ABB RobotStudio station: Assignment1 - Sela Shapira.rspag

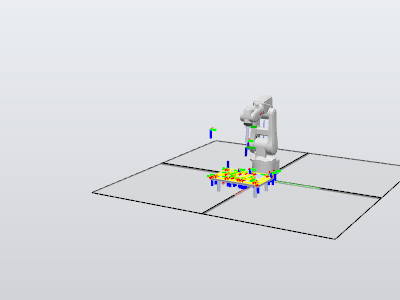
--- station ---
Station Assignment1 - Sela Shapira (saved by RobotStudio 23.2.10478.1)
Controller IRB120_3_58
  mechanical unit ROB_1: IRB120_3_58__01, 6 joints, base frame (0, 0, 0) mm
Layout (positions relative to the parent item):
  - IRB120_3_58__01 [mechanism, from %ABB.RobotStudio.Models.IRB120%\IRB120_3_58_G_01.rslib] at (0, 0, 0) mm; joint values [0.0316, -0.0225, 0.1697, 0.0059, 1.2834, -0.0224] (rad or m)
  - MyPen [mechanism, from Robotstudio\MyPen.rslib] at (312.81, 10.28, 513.58) mm, rotated rx 179.85 ry 8.04 rz -176.99 deg
  - A3 table [part] at (370, 0, 100) mm, rotated rx 90 ry 0 rz 90 deg, size 420 x 110 x 300 mm
  - Part_2 [part] at (370, 0, 100) mm, rotated rx 90 ry 0 rz 90 deg, size 420 x 0 x 300 mm
  - MDX_2 [part] at (370, 0, 115) mm, rotated rx 0 ry 0 rz -90 deg, size 400 x 260 x 10 mm
Attachment: MyPen is attached to IRB120_3_58__01 / Link6
Targets, tools, work objects and paths stored in the station and not in the controller backup, written as RAPID:
! task T_ROB1
MODULE Module1
  CONST robtarget Target_10:=[[0,0,0],[0,1,0,0],[0,0,0,0],[9E+09,9E+09,9E+09,9E+09,9E+09,9E+09]];
  CONST robtarget p2:=[[35.46,435.21,55.91],[0.0745505,-0.368836,0.926226,0.0225366],[0,-1,-1,0],[9E+09,9E+09,9E+09,9E+09,9E+09,9E+09]];
  CONST robtarget p3:=[[63.22,410.76,45.5],[0.0601149,-0.369349,0.92728,0.0109655],[0,-1,-1,0],[9E+09,9E+09,9E+09,9E+09,9E+09,9E+09]];
  CONST robtarget p4:=[[74.6,238.44,53.1],[0.0829113,-0.347129,0.933861,-0.0230488],[0,-1,-1,0],[9E+09,9E+09,9E+09,9E+09,9E+09,9E+09]];
  CONST robtarget p5:=[[80.38,145.13,41.2],[0.0559358,-0.237971,0.969261,-0.0278121],[-1,0,-1,0],[9E+09,9E+09,9E+09,9E+09,9E+09,9E+09]];
ENDMODULE


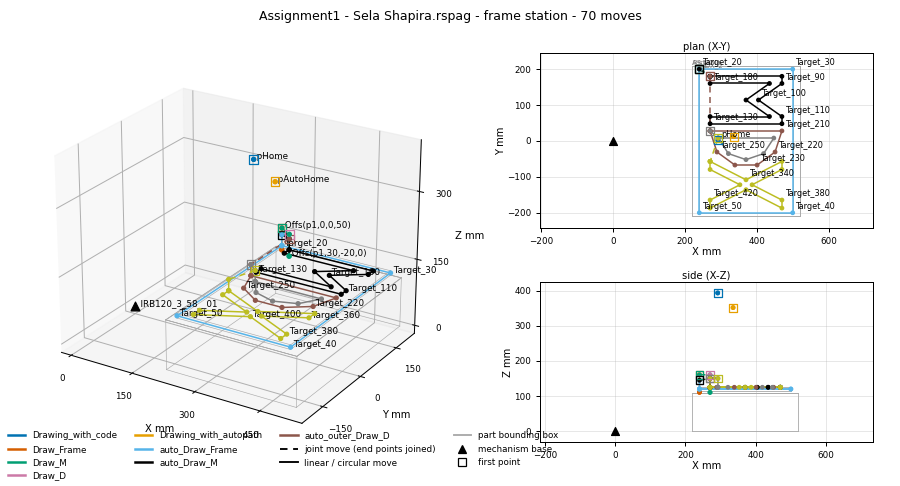
[picture p0: tool path of Assignment1 - Sela Shapira.rspag in frame station, 70 of 108 moves have a stored position in this frame; points joined in program order, loops and branches not executed]
--- Controller Data/IRB120_3_58/RAPID/TASK1/PROGMOD/CalibData.mod ---
MODULE CalibData
    TASK PERS wobjdata A3_paper:=[FALSE,TRUE,"",[[0,0,0],[1,0,0,0]],[[210.110012078,-230,0.978750149],[0.999999814,0.000539637,-0.000284188,0.000000153]]];
    TASK PERS tooldata MyPen:=[TRUE,[[0,0,163.48],[1,0,0,0]],[1,[0,0,1],[1,0,0,0],0,0,0]];
    TASK PERS wobjdata A3_table:=[FALSE,TRUE,"",[[0,0,0],[1,0,0,0]],[[220.46199678,-210,109.933409449],[0.999999726,0.000740141,0.000024177,-0.000000018]]];
ENDMODULE

--- Controller Data/IRB120_3_58/RAPID/TASK1/PROGMOD/Module1.mod ---
MODULE Module1
	CONST robtarget pHome:=[[291.94,1.72,393.38],[0.00283462,0.0189709,-0.999798,0.00597625],[0,-1,-1,0],[9E+09,9E+09,9E+09,9E+09,9E+09,9E+09]];
    CONST robtarget pAutoHome:=[[115.14,222.28,241.45],[0.0700142,-0.0263396,0.997195,0.00244358],[0,0,-1,0],[9E+09,9E+09,9E+09,9E+09,9E+09,9E+09]];
	CONST robtarget p1:=[[19.537513782,410.014448377,0.0],[0.00570496,-0.370161,0.928947,-0.00239576],[0,-1,-1,0],[9E+9,9E+9,9E+9,9E+9,9E+9,9E+9]];
    CONST robtarget Target_20:=[[19.537513782,410.014448377,9.460553594],[0,1,0,0],[0,-1,-2,0],[9E+09,9E+09,9E+09,9E+09,9E+09,9E+09]];
    CONST robtarget Target_30:=[[279.537531526,410.014489539,9.473159734],[0,1,0,0],[0,0,-2,0],[9E+09,9E+09,9E+09,9E+09,9E+09,9E+09]];
    CONST robtarget Target_40:=[[279.537531641,10.014893228,10.065272423],[0,1,0,0],[-1,0,-3,0],[9E+09,9E+09,9E+09,9E+09,9E+09,9E+09]];
    CONST robtarget Target_50:=[[19.537516435,10.014891835,10.052721434],[0,1,0,0],[-1,0,-3,0],[9E+09,9E+09,9E+09,9E+09,9E+09,9E+09]];
    CONST robtarget Target_60:=[[19.537516351,410.014453588,9.460608796],[0,1,0,0],[0,0,-2,0],[9E+09,9E+09,9E+09,9E+09,9E+09,9E+09]];
    CONST robtarget Target_70:=[[49.537291728,390.021897691,14.491613569],[0,1,0,0],[0,-1,-2,0],[9E+09,9E+09,9E+09,9E+09,9E+09,9E+09]];
    CONST robtarget Target_80:=[[249.537269612,390.021892362,14.50128376],[0,1,0,0],[0,0,-2,0],[9E+09,9E+09,9E+09,9E+09,9E+09,9E+09]];
    CONST robtarget Target_90:=[[249.53727432,370.021915332,14.530935987],[0,1,0,0],[0,0,-2,0],[9E+09,9E+09,9E+09,9E+09,9E+09,9E+09]];
    CONST robtarget Target_100:=[[184.253140009,324.008160862,14.595892622],[0,1,0,0],[0,0,-2,0],[9E+09,9E+09,9E+09,9E+09,9E+09,9E+09]];
    CONST robtarget Target_110:=[[249.537267147,277.994418069,14.667111324],[0,1,0,0],[0,0,-2,0],[9E+09,9E+09,9E+09,9E+09,9E+09,9E+09]];
    CONST robtarget Target_120:=[[249.537274344,257.994437677,14.696768382],[0,1,0,0],[0,0,-2,0],[9E+09,9E+09,9E+09,9E+09,9E+09,9E+09]];
    CONST robtarget Target_130:=[[49.537289789,257.994422788,14.687052106],[-0.000000001,1,0.000000021,-0.000000007],[0,0,-2,0],[9E+09,9E+09,9E+09,9E+09,9E+09,9E+09]];
    CONST robtarget Target_140:=[[49.537274573,277.994401407,14.657491958],[0,1,0,0],[0,0,-2,0],[9E+09,9E+09,9E+09,9E+09,9E+09,9E+09]];
    CONST robtarget Target_150:=[[214.821376774,277.994415341,14.665431207],[0,1,0,0],[0,0,-2,0],[9E+09,9E+09,9E+09,9E+09,9E+09,9E+09]];
    CONST robtarget Target_160:=[[149.537271511,324.008157847,14.594164036],[-0.000000007,1,0.000000048,-0.000000022],[0,0,-2,0],[9E+09,9E+09,9E+09,9E+09,9E+09,9E+09]];
    CONST robtarget Target_170:=[[214.821408758,370.02191284,14.529257337],[0,1,0,0],[0,0,-2,0],[9E+09,9E+09,9E+09,9E+09,9E+09,9E+09]];
    CONST robtarget Target_180:=[[49.53728079,370.021897613,14.521217152],[-0.000000009,1,0.000000018,-0.000000015],[0,0,-2,0],[9E+09,9E+09,9E+09,9E+09,9E+09,9E+09]];
    CONST robtarget Target_190:=[[49.53727455,390.021879062,14.491659563],[0,1,0,0],[0,0,-2,0],[9E+09,9E+09,9E+09,9E+09,9E+09,9E+09]];
    CONST robtarget Target_200:=[[49.537288263,237.994446649,14.716657267],[0,1,0,0],[0,-1,-2,0],[9E+09,9E+09,9E+09,9E+09,9E+09,9E+09]];
    CONST robtarget Target_210:=[[249.537277298,237.994460289,14.726342327],[0,1,0,0],[0,0,-2,0],[9E+09,9E+09,9E+09,9E+09,9E+09,9E+09]];
    CONST robtarget Target_220:=[[230.438959272,179.215991889,14.812410932],[0.000000001,1,0.000000022,-0.000000014],[-1,0,-3,0],[9E+09,9E+09,9E+09,9E+09,9E+09,9E+09]];
    CONST robtarget Target_230:=[[180.438990665,142.888893103,14.863780968],[-0.000000003,1,0.000000029,0.000000018],[-1,0,-3,0],[9E+09,9E+09,9E+09,9E+09,9E+09,9E+09]];
    CONST robtarget Target_240:=[[118.635575084,142.888902762,14.860827544],[0,1,0,0],[-1,0,-3,0],[9E+09,9E+09,9E+09,9E+09,9E+09,9E+09]];
    CONST robtarget Target_250:=[[68.635575135,179.215985772,14.804635469],[0,1,0,0],[-1,0,-3,0],[9E+09,9E+09,9E+09,9E+09,9E+09,9E+09]];
    CONST robtarget Target_260:=[[49.537274582,237.994445231,14.716703222],[0,1,0,0],[0,0,-2,0],[9E+09,9E+09,9E+09,9E+09,9E+09,9E+09]];
    CONST robtarget Target_270:=[[72.077604833,217.994469382,14.74735851],[0,1,0,0],[0,-1,-2,0],[9E+09,9E+09,9E+09,9E+09,9E+09,9E+09]];
    CONST robtarget Target_280:=[[226.996972617,217.994479605,14.754844037],[0,1,0,0],[0,0,-2,0],[9E+09,9E+09,9E+09,9E+09,9E+09,9E+09]];
    CONST robtarget Target_290:=[[198.527081303,174.748975342,14.817484944],[0.000000001,1,0,-0.000000012],[-1,0,-3,0],[9E+09,9E+09,9E+09,9E+09,9E+09,9E+09]];
    CONST robtarget Target_300:=[[149.537285205,157.994535259,14.839916567],[0,1,0.000000033,-0.000000003],[-1,0,-3,0],[9E+09,9E+09,9E+09,9E+09,9E+09,9E+09]];
    CONST robtarget Target_310:=[[100.547479679,174.748964983,14.812790995],[0,1,0,0],[-1,0,-3,0],[9E+09,9E+09,9E+09,9E+09,9E+09,9E+09]];
    CONST robtarget Target_320:=[[72.077587245,217.99446886,14.747346368],[0,1,-0.000000005,0],[0,0,-2,0],[9E+09,9E+09,9E+09,9E+09,9E+09,9E+09]];
    CONST robtarget Target_330:=[[49.537287698,152.994536899,14.84247854],[0,1,0,0],[-1,0,-2,0],[9E+09,9E+09,9E+09,9E+09,9E+09,9E+09]];
    CONST robtarget Target_340:=[[149.537280469,101.772303848,14.923138018],[0,1,0,0],[-1,0,-3,0],[9E+09,9E+09,9E+09,9E+09,9E+09,9E+09]];
    CONST robtarget Target_350:=[[249.537274366,152.994552716,14.852197949],[0,1,0,0],[-1,0,-3,0],[9E+09,9E+09,9E+09,9E+09,9E+09,9E+09]];
    CONST robtarget Target_360:=[[249.537281332,130.523514119,14.885415007],[0,1,0,0],[-1,0,-3,0],[9E+09,9E+09,9E+09,9E+09,9E+09,9E+09]];
    CONST robtarget Target_370:=[[166.509079524,87.994622174,14.944366822],[0,1,-0.000000013,0],[-1,0,-3,0],[9E+09,9E+09,9E+09,9E+09,9E+09,9E+09]];
    CONST robtarget Target_380:=[[249.53727951,45.465764096,15.011316491],[0,1,0,0],[-1,0,-3,0],[9E+09,9E+09,9E+09,9E+09,9E+09,9E+09]];
    CONST robtarget Target_390:=[[249.537270203,22.994699855,15.044601216],[0,1,0,0],[-1,0,-3,0],[9E+09,9E+09,9E+09,9E+09,9E+09,9E+09]];
    CONST robtarget Target_400:=[[149.537274499,74.216884509,14.963975803],[0,1,0,0],[-1,0,-3,0],[9E+09,9E+09,9E+09,9E+09,9E+09,9E+09]];
    CONST robtarget Target_410:=[[49.537288239,22.99466738,15.0349256],[0,1,0.00000001,0],[-1,0,-3,0],[9E+09,9E+09,9E+09,9E+09,9E+09,9E+09]];
    CONST robtarget Target_420:=[[49.537274622,45.465721269,15.00170026],[0,1,0,0],[-1,0,-3,0],[9E+09,9E+09,9E+09,9E+09,9E+09,9E+09]];
    CONST robtarget Target_430:=[[132.56551457,87.994615534,14.942760205],[0,1,0,0],[-1,0,-3,0],[9E+09,9E+09,9E+09,9E+09,9E+09,9E+09]];
    CONST robtarget Target_440:=[[49.537274604,130.523497879,14.875790661],[0,1,0,0],[-1,0,-3,0],[9E+09,9E+09,9E+09,9E+09,9E+09,9E+09]];
    CONST robtarget Target_450:=[[49.5372746,152.994538359,14.842527157],[0,1,0,0],[-1,0,-3,0],[9E+09,9E+09,9E+09,9E+09,9E+09,9E+09]];
    !***********************************************************
    !
    ! Module:  Module1
    !
    ! Description:
    !   <Insert description here>
    !
    ! Author: selas
    !
    ! Version: 1.0
    !
    !***********************************************************


    !***********************************************************
    !
    ! Procedure main
    !
    !   This is the entry point of your program
    !
    !***********************************************************

    ! ============ Variables For Draw_M ===============
    VAR num Letter_M_Height:= 200;
    VAR num mid_Letter_M_Height:= 100;
    VAR num Letter_M_Width:= 132.03;
    VAR num Letter_M_thickness:= 20;
    VAR num Letter_M_bigpeack:= 65.28;
    VAR num Letter_M_smallpeack:= 34.72;
    VAR num MidLetter:= 66.015;
    ! ============ Variables For Draw_D ===============
    VAR num Letter_D_Height:= 200;
    VAR num InnerLetter_D_Height:= 160;
    VAR num Outer_D_Radius:= 100;
    VAR num Inner_D_radius:= 80;
    VAR num Letter_D_distance:= 152.03;
    VAR num mid_Letter_D_Height:= 100;
    VAR num InnerLetter_D_distance:= 172.03;
    VAR num Letter_D_thickness:= 20;
    ! ============ Variables For Draw_X ===============
    VAR num Letter_X_Height:= 200;
    VAR num Letter_X_thickness:= 20;
    VAR num Letter_X_distance:= 237.03;
    VAR num Letter_X_Width:= 130.0;
    VAR num Letter_X_peack:= 83.03;
    VAR num MidLetterX:= 65;
    VAR num Letter_X_midpeack:= 51.22;
    VAR num Letter_X_leg:= 22.47;
    VAR num mid_Letter_X_Height:= 100;


    PROC main()
        VAR num answer:= 0;
        TPreadFK answer, "which method would you like to draw", "code", "autopath", stEmpty, stEmpty,stEmpty;
        IF answer = 1 THEN
            Drawing_with_code;
        ELSEIF answer = 2 THEN
            Drawing_with_autopath;
        ELSE
        ENDIF
    ENDPROC

    PROC Drawing_with_code()
        MoveJ pHome, v300, fine, MyPen;
        Draw_Frame 400, 260;
        Draw_M;
        Draw_D;
        Draw_X;
        MoveJ pHome, v300, fine, MyPen;
    ENDPROC

	PROC Draw_Frame(num Length, num Width)
        MoveJ Offs(p1, 0, 0, 50),v200,fine,MyPen\WObj:=A3_table;
        MoveL Offs(p1, 0, 0, 0),v200,fine,MyPen\WObj:=A3_table;
        MoveL Offs(p1, Width, 0, 0), v800, fine, MyPen\WObj:=A3_table;
        MoveL Offs(p1, Width, -Length, 0), v800, fine, MyPen\WObj:=A3_table;
        MoveL Offs(p1, 0, -Length, 0), v800, fine, MyPen\WObj:=A3_table;
        MoveL Offs(p1, 0, 0, 0), v800, fine, MyPen\WObj:=A3_table;
	ENDPROC
    PROC Draw_M()
        MoveL Offs(p1, 0, 0, 50),v200,fine,MyPen\WObj:=A3_table;
        MoveJ Offs(p1, 30, -20, 50),v200,fine,MyPen\WObj:=A3_table;
        MoveL Offs(p1, 30, -20, 0),v200,fine,MyPen\WObj:=A3_table;
        MoveL Offs(p1, 30+Letter_M_Height, -20, 0),v800,fine,MyPen\WObj:=A3_table;
        MoveL Offs(p1, 30+Letter_M_Height, -20-Letter_M_thickness, 0),v800,fine,MyPen\WObj:=A3_table;
        MoveL Offs(p1, 30+Letter_M_Height-Letter_M_bigpeack, -20-MidLetter, 0),v800,fine,MyPen\WObj:=A3_table;
        MoveL Offs(p1, 30+Letter_M_Height, -20-Letter_M_Width+Letter_M_thickness, 0),v800,fine,MyPen\WObj:=A3_table;
        MoveL Offs(p1, 30+Letter_M_Height, -20-Letter_M_Width, 0),v800,fine,MyPen\WObj:=A3_table;
        MoveL Offs(p1, 30, -20-Letter_M_Width, 0),v800,fine,MyPen\WObj:=A3_table;
        MoveL Offs(p1, 30, -20-Letter_M_Width+Letter_M_thickness, 0),v800,fine,MyPen\WObj:=A3_table;
        MoveL Offs(p1, 30+Letter_M_Height-Letter_M_smallpeack, -20-Letter_M_Width+Letter_M_thickness, 0),v800,fine,MyPen\WObj:=A3_table;
        MoveL Offs(p1, 30+mid_Letter_M_Height, -20-MidLetter, 0),v800,fine,MyPen\WObj:=A3_table;
        MoveL Offs(p1, 30+Letter_M_Height-Letter_M_smallpeack, -20-Letter_M_thickness, 0),v800,fine,MyPen\WObj:=A3_table;
        MoveL Offs(p1, 30, -20-Letter_M_thickness, 0),v800,fine,MyPen\WObj:=A3_table;
        MoveJ Offs(p1, 30, -20, 0),v800,fine,MyPen\WObj:=A3_table;
        WaitTime 0.2;
    ENDPROC
    PROC Draw_D()
        MoveL Offs(p1, 30, -20, 50),v200,fine,MyPen\WObj:=A3_table;
        MoveJ Offs(p1, 30, -20-Letter_D_distance, 50),v200,fine,MyPen\WObj:=A3_table;
        MoveL Offs(p1, 30, -20-Letter_D_distance, 0),v200,fine,MyPen\WObj:=A3_table;
        MoveL Offs(p1, 30+Letter_D_Height, -20-Letter_D_distance, 0),v800,fine,MyPen\WObj:=A3_table;
        MoveC Offs(p1, 30+mid_Letter_D_Height, -20-Letter_D_distance-Outer_D_Radius, 0),Offs(p1, 30, -20-Letter_D_distance ,0),v800,fine,MyPen\WObj:=A3_table;
        MoveL Offs(p1, 30, -20-Letter_D_distance, 50),v200,fine,MyPen\WObj:=A3_table;
        MoveJ Offs(p1, 30+Letter_D_thickness, -20-InnerLetter_D_distance, 50),v200,fine,MyPen\WObj:=A3_table;
        MoveL Offs(p1, 30+Letter_D_thickness, -20-InnerLetter_D_distance, 0),v200,fine,MyPen\WObj:=A3_table;
        MoveL Offs(p1, 30+InnerLetter_D_Height, -20-InnerLetter_D_distance, 0),v800,fine,MyPen\WObj:=A3_table;
        MoveC Offs(p1, 30+mid_Letter_D_Height, -20-Letter_D_distance-Inner_D_radius, 0),Offs(p1, 30+Letter_D_thickness, -20-InnerLetter_D_distance ,0),v800,fine,MyPen\WObj:=A3_table;
        WaitTime 0.2;
    ENDPROC
    PROC Draw_X()
        MoveL Offs(p1, 30+Letter_D_thickness, -20-InnerLetter_D_distance, 50),v200,fine,MyPen\WObj:=A3_table;
        MoveJ Offs(p1, 30, -20-Letter_X_distance, 50),v200,fine,MyPen\WObj:=A3_table;
        MoveL Offs(p1, 30, -20-Letter_X_distance, 0),v200,fine,MyPen\WObj:=A3_table;
        MoveL Offs(p1, 30+mid_Letter_X_Height, -20-Letter_X_distance-Letter_X_midpeack, 0),v800,fine,MyPen\WObj:=A3_table;
        MoveL Offs(p1, 30+Letter_X_Height, -20-Letter_X_distance, 0),v800,fine,MyPen\WObj:=A3_table;
        MoveL Offs(p1, 30+Letter_X_Height, -20-Letter_X_distance-Letter_X_leg, 0),v800,fine,MyPen\WObj:=A3_table;
        MoveL Offs(p1, 30+Letter_X_Height-Letter_X_peack, -20-Letter_X_distance-MidLetterX, 0),v800,fine,MyPen\WObj:=A3_table;
        MoveL Offs(p1, 30+Letter_X_Height, -20-Letter_X_distance-Letter_X_Width+Letter_X_leg, 0),v800,fine,MyPen\WObj:=A3_table;
        MoveL Offs(p1, 30+Letter_X_Height, -20-Letter_X_distance-Letter_X_Width, 0),v800,fine,MyPen\WObj:=A3_table;
        MoveL Offs(p1, 30+mid_Letter_X_Height, -20-Letter_X_distance-Letter_X_Width+Letter_X_midpeack, 0),v800,fine,MyPen\WObj:=A3_table;
        MoveL Offs(p1, 30, -20-Letter_X_distance-Letter_X_Width, 0),v800,fine,MyPen\WObj:=A3_table;
        MoveL Offs(p1, 30, -20-Letter_X_distance-Letter_X_Width+Letter_X_leg, 0),v800,fine,MyPen\WObj:=A3_table;
        MoveL Offs(p1, 30+Letter_X_peack, -20-Letter_X_distance-MidLetterX, 0),v800,fine,MyPen\WObj:=A3_table;
        MoveL Offs(p1, 30, -20-Letter_X_distance-Letter_X_leg, 0),v800,fine,MyPen\WObj:=A3_table;
        MoveL Offs(p1, 30, -20-Letter_X_distance, 0),v800,fine,MyPen\WObj:=A3_table;
        WaitTime 0.2;
    ENDPROC

    PROC Drawing_with_autopath()
        MoveJ pAutoHome, v300, fine, MyPen\WObj:=A3_table;
        auto_Draw_Frame;
        auto_Draw_M;
        auto_outer_Draw_D;
        auto_inner_Draw_D;
        auto_Draw_X;
        MoveJ pAutoHome, v300, fine, MyPen\WObj:=A3_table;
    ENDPROC

    PROC auto_Draw_Frame()
        MoveJ Offs(Target_20, 0, 0, 25),v200,fine,MyPen\WObj:=A3_table;
        MoveL Offs(Target_20, 0, 0, 0),v200,fine,MyPen\WObj:=A3_table;
        MoveL Target_20,v1000,fine,MyPen\WObj:=A3_table;
        MoveL Target_30,v1000,fine,MyPen\WObj:=A3_table;
        MoveL Target_40,v1000,fine,MyPen\WObj:=A3_table;
        MoveL Target_50,v1000,fine,MyPen\WObj:=A3_table;
        MoveL Target_60,v1000,fine,MyPen\WObj:=A3_table;
    ENDPROC
    PROC auto_Draw_M()
        MoveL Offs(Target_20, 0, 0, 25),v200,fine,MyPen\WObj:=A3_table;
        MoveJ Offs(Target_70, 0, 0, 25),v200,fine,MyPen\WObj:=A3_table;
        MoveL Offs(Target_70, 0, 0, 0),v200,fine,MyPen\WObj:=A3_table;
        MoveL Target_70,v1000,fine,MyPen\WObj:=A3_table;
        MoveL Target_80,v1000,fine,MyPen\WObj:=A3_table;
        MoveL Target_90,v1000,fine,MyPen\WObj:=A3_table;
        MoveL Target_100,v1000,fine,MyPen\WObj:=A3_table;
        MoveL Target_110,v1000,fine,MyPen\WObj:=A3_table;
        MoveL Target_120,v1000,fine,MyPen\WObj:=A3_table;
        MoveL Target_130,v1000,fine,MyPen\WObj:=A3_table;
        MoveL Target_140,v1000,fine,MyPen\WObj:=A3_table;
        MoveL Target_150,v1000,fine,MyPen\WObj:=A3_table;
        MoveL Target_160,v1000,fine,MyPen\WObj:=A3_table;
        MoveL Target_170,v1000,fine,MyPen\WObj:=A3_table;
        MoveL Target_180,v1000,fine,MyPen\WObj:=A3_table;
        MoveL Target_190,v1000,fine,MyPen\WObj:=A3_table;
    ENDPROC
    PROC auto_outer_Draw_D()
        MoveL Offs(Target_70, 0, 0, 25),v200,fine,MyPen\WObj:=A3_table;
        MoveJ Offs(Target_200, 0, 0, 25),v200,fine,MyPen\WObj:=A3_table;
        MoveL Offs(Target_200, 0, 0, 0),v200,fine,MyPen\WObj:=A3_table;
        MoveL Target_200,v1000,fine,MyPen\WObj:=A3_table;
        MoveL Target_210,v1000,fine,MyPen\WObj:=A3_table;
        MoveL Target_220,v1000,z200,MyPen\WObj:=A3_table;
        MoveL Target_230,v1000,z200,MyPen\WObj:=A3_table;
        MoveL Target_240,v1000,z200,MyPen\WObj:=A3_table;
        MoveL Target_250,v1000,z200,MyPen\WObj:=A3_table;
        MoveL Target_260,v1000,z200,MyPen\WObj:=A3_table;
    ENDPROC
    PROC auto_inner_Draw_D()
        MoveL Offs(Target_200, 0, 0, 25),v200,fine,MyPen\WObj:=A3_table;
        MoveJ Offs(Target_270, 0, 0, 25),v200,fine,MyPen\WObj:=A3_table;
        MoveL Offs(Target_270, 0, 0, 0),v200,fine,MyPen\WObj:=A3_table;
        MoveL Target_270,v1000,fine,MyPen\WObj:=A3_table;
        MoveL Target_280,v1000,fine,MyPen\WObj:=A3_table;
        MoveL Target_290,v1000,z100,MyPen\WObj:=A3_table;
        MoveL Target_300,v1000,z100,MyPen\WObj:=A3_table;
        MoveL Target_310,v1000,z100,MyPen\WObj:=A3_table;
        MoveL Target_320,v1000,z100,MyPen\WObj:=A3_table;
    ENDPROC
    PROC auto_Draw_X()
        MoveL Offs(Target_270, 0, 0, 25),v200,fine,MyPen\WObj:=A3_table;
        MoveJ Offs(Target_330, 0, 0, 25),v200,fine,MyPen\WObj:=A3_table;
        MoveL Offs(Target_330, 0, 0, 0),v200,fine,MyPen\WObj:=A3_table;
        MoveL Target_330,v1000,fine,MyPen\WObj:=A3_table;
        MoveL Target_340,v1000,fine,MyPen\WObj:=A3_table;
        MoveL Target_350,v1000,fine,MyPen\WObj:=A3_table;
        MoveL Target_360,v1000,fine,MyPen\WObj:=A3_table;
        MoveL Target_370,v1000,fine,MyPen\WObj:=A3_table;
        MoveL Target_380,v1000,fine,MyPen\WObj:=A3_table;
        MoveL Target_390,v1000,fine,MyPen\WObj:=A3_table;
        MoveL Target_400,v1000,fine,MyPen\WObj:=A3_table;
        MoveL Target_410,v1000,fine,MyPen\WObj:=A3_table;
        MoveL Target_420,v1000,fine,MyPen\WObj:=A3_table;
        MoveL Target_430,v1000,fine,MyPen\WObj:=A3_table;
        MoveL Target_440,v1000,fine,MyPen\WObj:=A3_table;
        MoveL Target_450,v1000,fine,MyPen\WObj:=A3_table;
    ENDPROC
ENDMODULE
